(* PLC project  *)

PROGRAM P

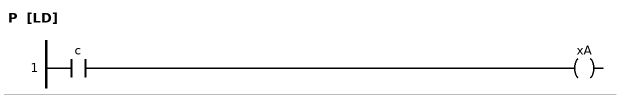
(* LD diagram, written out as Structured Text *)
xA := c;
END_PROGRAM
